// TIA Portal V16 export
// export: Created 2022-03-28T07:44:08.1425643Z, ExportSetting WithDefaults, DisplayName Totally Integrated Automation Portal, DisplayVersion V16 Update 5, DisplayName TIA Portal Version Control Interface, DisplayVersion V16 Update 2, DisplayName TIA Portal Openness, DisplayVersion V16 Update 5, DisplayName STEP 7 Professional, DisplayVersion V16 Update 5, DisplayName STEP 7 Safety, DisplayVersion V16, DisplayName WinCC Professional, DisplayVersion V16 Update 5
VAR_GLOBAL   // PLC tag table "Tabla de variables estándar"
   System_Byte AT %MB1001 : Byte;
   FirstScan AT %M1001.0 : Bool;
   DiagStatusUpdate AT %M1001.1 : Bool;
   AlwaysTRUE AT %M1001.2 : Bool;
   AlwaysFALSE AT %M1001.3 : Bool;
   Clock_Byte AT %MB1000 : Byte;
   Clock_10Hz AT %M1000.0 : Bool;
   Clock_5Hz AT %M1000.1 : Bool;
   "Clock_2.5Hz" AT %M1000.2 : Bool;
   Clock_2Hz AT %M1000.3 : Bool;
   "Clock_1.25Hz" AT %M1000.4 : Bool;
   Clock_1Hz AT %M1000.5 : Bool;
   "Clock_0.625Hz" AT %M1000.6 : Bool;
   "Clock_0.5Hz" AT %M1000.7 : Bool;
   Tag_1 AT %MW100 : Word;
   Tag_2 AT %M10.0 : Bool;
   bStartShortBolt AT %M20.0 : Bool;
   bStartMediumBolt AT %M20.1 : Bool;
   bStartLongBolt AT %M20.2 : Bool;
   bStartWeldingGripper_3 AT %M20.3 : Bool;
   bRetractGripper_3 AT %M20.4 : Bool;
   Tag_8 AT %M20.5 : Bool;
   Tag_9 AT %M20.6 : Bool;
   Tag_10 AT %M20.7 : Bool;
   bGripper_3_Conditions AT %M29.0 : Bool;
   bStartSmallNut AT %M21.0 : Bool;
   bStartBigNut AT %M21.1 : Bool;
   bStartWeldingGripper_2 AT %M21.2 : Bool;
   bRetractGripper_2 AT %M21.3 : Bool;
   Tag_16 AT %M21.4 : Bool;
   Tag_17 AT %M21.5 : Bool;
   Tag_18 AT %M21.6 : Bool;
   Tag_19 AT %M21.7 : Bool;
   bGripper_2_Conditions AT %M29.1 : Bool;
   bStartSpot AT %M22.0 : Bool;
   bStartWeldingGripper_1 AT %M22.1 : Bool;
   bRetractGripper_1 AT %M22.2 : Bool;
   Tag_24 AT %M22.3 : Bool;
   Tag_25 AT %M22.4 : Bool;
   Tag_26 AT %M22.5 : Bool;
   Tag_27 AT %M22.6 : Bool;
   Tag_28 AT %M22.7 : Bool;
   bGripper_1_Conditions AT %M29.2 : Bool;
   bCycleConditions AT %M29.3 : Bool;
   bEndOfCycle AT %M23.0 : Bool;
   bWeldingNOK AT %M23.1 : Bool;
   bToScrap AT %M23.2 : Bool;
   bScraped AT %M23.3 : Bool;
   bScrapBoxFull AT %M23.4 : Bool;
   bConsecutiveNOKtoBlock AT %M23.5 : Bool;
   bRobotAuto AT %M23.6 : Bool;
   bProductionCompleted AT %M23.7 : Bool;
   bAction_1 AT %M24.0 : Bool;
   bAction_2 AT %M24.1 : Bool;
   bAction_3 AT %M24.2 : Bool;
   bAction_4 AT %M24.3 : Bool;
   bAction_5 AT %M24.4 : Bool;
   bAction_6 AT %M24.5 : Bool;
   bEndSequence AT %M24.6 : Bool;
   BWelderProgNumber AT %MB12 : Byte;
   bWelderProg_Bit_0 AT %M12.0 : Bool;
   bWelderProg_Bit_1 AT %M12.1 : Bool;
   bWelderProg_Bit_2 AT %M12.2 : Bool;
   bWelderProg_Bit_3 AT %M12.3 : Bool;
   bWelderProg_Bit_4 AT %M12.4 : Bool;
   Tag_53 AT %MW20 : Int;
   Tag_54 AT %MW22 : Int;
   Tag_55 AT %MW24 : Int;
   "Alarmes 1" AT %MW200 : Word;
   "Alarmes 2" AT %MW202 : Word;
   bAnyAlarm AT %M210.0 : Bool;
   Tag_59 AT %MD200 : DWord;
   bEmergenciesNOK AT %M200.0 : Bool;
   bPressureFault AT %M200.1 : Bool;
   bFlowFault AT %M200.2 : Bool;
   "Alarma barrera cajon rechazo" AT %M200.3 : Bool;
   "Alarma pinza 1 no avanza" AT %M201.0 : Bool;
   "Alarma pinza 1 No retrocede" AT %M201.1 : Bool;
   "Alarma pinza 2 No avanza" AT %M201.2 : Bool;
   "Alarma pinza 2 No retrocede" AT %M201.3 : Bool;
   "Alarma pinza3 no avanza" AT %M201.4 : Bool;
   "Alarma pinza 3 No retrocede" AT %M201.5 : Bool;
   bWelderNotReady AT %M200.4 : Bool;
   bWelderNotResponding AT %M200.5 : Bool;
   "Alarma barrera obstruida" AT %M202.0 : Bool;
   Tag_73 AT %M200.6 : Bool;
   "Aviso perno corto incorreto" AT %M202.1 : Bool;
   "Aviso perno medio incorrecto" AT %M202.2 : Bool;
   "Aviso perno largo incorrecto" AT %M202.3 : Bool;
   "Aviso pieza mala" AT %M202.4 : Bool;
   "Aviso tirar pieza mala" AT %M202.5 : Bool;
   Tag_79 AT %M202.6 : Bool;
   bInitConditions AT %M29.4 : Bool;
   "Alarmes 6" AT %MW210 : Word;
   Tag_56 AT %M200.7 : Bool;
   Tag_57 AT %M5.0 : Bool;
   Tag_60 AT %M5.1 : Bool;
   Tag_61 AT %M5.2 : Bool;
   Tag_62 AT %M5.3 : Bool;
   Tag_63 AT %M5.4 : Bool;
   Tag_64 AT %M5.5 : Bool;
   Tag_58 AT %M7.0 : Bool;
   Tag_65 AT %M6.5 : Bool;
   Tag_66 AT %M6.4 : Bool;
   Tag_67 AT %M6.2 : Bool;
   Tag_68 AT %M6.3 : Bool;
   Tag_69 AT %M6.0 : Bool;
   Tag_70 AT %M6.1 : Bool;
   bTemp_PAP AT %M100.0 : Bool;
   bRedLamp_3_NonInverted AT %M50.0 : Bool;
   bRedLamp_1_Inverted AT %M50.1 : Bool;
   bAmberLamp_3_NonInverted AT %M50.2 : Bool;
   bGreenLamp_3_NonInverted AT %M50.4 : Bool;
   bAmberLamp_1_Inverted AT %M50.3 : Bool;
   bGreenLamp_1_Inverted AT %M50.5 : Bool;
   bRedLamp_1_NonInverted AT %M50.6 : Bool;
   bRedLamp_3_Inverted AT %M50.7 : Bool;
   bAmberLamp_1_NonInverted AT %M51.0 : Bool;
   bAmberLamp_3_Inverted AT %M51.1 : Bool;
   bGreenLamp_1_NonInverted AT %M51.2 : Bool;
   bGreenLamp_3_Inverted AT %M51.3 : Bool;
   bStartLamp_1_NonInverted AT %M51.4 : Bool;
   bStartLamp_3_NonInverted AT %M51.5 : Bool;
   bStartLamp_3_Inverted AT %M51.6 : Bool;
   bStartLamp_1_Inverted AT %M51.7 : Bool;
   bGripper_3_NonInverted AT %M52.0 : Bool;
   bGripper_1_NonInverted AT %M52.1 : Bool;
   bGripper_3_Inverted AT %M52.3 : Bool;
   bGripper_1_Inverted AT %M52.2 : Bool;
END_VAR
